Fanuc KAREL source: kt00004.KL

-- PROVISIONAL review KL for V1013-1; original PC SHA256 d5725a2d66bf454d601817318aafe2d693e8f23face0300a6c75dd369a482001
-- Incomplete behavior may be omitted. Consult companion uncertainty JSON. Do not deploy.
PROGRAM KT00004
%NOLOCKGROUP
VAR
  I1 : INTEGER
  R2 : REAL
  OUT : REAL
BEGIN
  -- UNRESOLVED_PC offsets 5-16; opcodes 2E,23
  -- UNRESOLVED_PC offsets 21-32; opcodes 2E,23
  -- UNRESOLVED_PC offsets 37-58; opcodes 21,21,29,64,69,23
  -- UNRESOLVED_PC offsets 63-67; opcodes 7F
END KT00004
